Staubli VAL3: Empilement.pgx

program Empilement()
  local point l_pPoint
  local point l_pPoint1
  local num l_CurrentLigne
  local num l_CurrentPiece
begin

  for l_CurrentLigne=0 to nLigne -1
    nDebut=clock()
    for l_CurrentPiece=0 to nPieceLigne -1
      trDecalPiece={l_CurrentLigne*nDistanceLigne,l_CurrentPiece*nDistancePiece,0,0,0,0}
      trDecalHauteur={l_CurrentLigne*nDistanceLigne,300,l_CurrentPiece*nHauteurPiece,0,0,0}
      l_pPoint=compose(pP1,world,trDecalPiece)
      l_pPoint1=compose(pP1,world,trDecalHauteur)
      call Prise(l_pPoint)
      call Pause(l_pPoint1)
    endFor
    nFin=clock()
    put("current ligne ")
    putln(l_CurrentLigne+1)
    put( " : " )
    putln( nFin-nDebut)
    put(" s")
    delay(2)
  endFor
  movej(jDepart,tPince,mRapide)


end
